FUNCTION TFGetEnableCode : ARRAY [1..MAXFORMINGCODE*MAXFORMING] OF INT
VAR_INPUT
	Forming : POINTER TO ARRAY [1..MAXFORMING] OF TFMachinePalletizer_Forming;
END_VAR
VAR
	EnableCode : ARRAY [1..MAXFORMINGCODE*MAXFORMING] OF INT;
	pp : UINT;
	pf : UINT;
	c : INT;
	i : UINT;
END_VAR

FOR i:=1 TO MAXFORMINGCODE*MAXFORMING DO
	EnableCode[i]:= 0;
END_FOR
c:=1; 
(* Per Tutte le Formature Attive *)
FOR pf:=1 TO MAXFORMING DO
	IF Forming^[pf].Enable = 1 THEN
		(* Per tutti i codici di Pallettizzazione Validi *)
		FOR pp:=1 TO MAXFORMINGCODE DO
			IF Forming^[pf].Code[pp] > 0 THEN
				EnableCode[c] := Forming^[pf].Code[pp];
				c := c+1;
			END_IF
		END_FOR
	END_IF
END_FOR
TFGetEnableCode := EnableCode;

END_FUNCTION

(* stored: Version 1.1.0.1, ProductVersion 3.1.4024.11
   POU TFGetEnableCode: Id {d2c90ea0-6893-4b60-a8d4-8bd31baf3ee1}, SpecialFunc None *)
